FUNCTION_BLOCK CreateRecipeFile
VAR_INPUT
END_VAR
VAR_OUTPUT
END_VAR
VAR
END_VAR

END_FUNCTION_BLOCK

(* stored: Version 1.1.0.1, ProductVersion 3.1.4022.18
   POU CreateRecipeFile: Id {21b267a5-cfef-492a-83c2-e2e2b8265fee}, SpecialFunc None *)
